PROGRAM MAIN
VAR
	fbTrafficLightController: FB_TrafficLightController;
	nNumTraffic: SINT := 4;
	bInitialized: BOOL := FALSE;
END_VAR

IF NOT bInitialized THEN
	bInitialized := TRUE;
	Setup();
END_IF

fbTrafficLightController();

METHOD PRIVATE Setup
fbTrafficLightController.NumberOfTrafficLights := nNumTraffic;
fbTrafficLightController.Setup(2, T#10S, T#3S, T#8S);
END_METHOD

END_PROGRAM

(* stored: Version 1.1.0.1, ProductVersion 3.1.4024.12
   POU MAIN: Id {14432245-9782-4d97-91be-5e69b86d0198}, SpecialFunc None
   Method Setup: Id {017bf35d-4b8b-424f-8833-172d4e6e6df5} *)
